FUNCTION_BLOCK FB_ParamMediatorWeu IMPLEMENTS I_ParamMediator
VAR
  _pCreateWorker : POINTER TO FB_WorkerDefGrid_Python;
  _pCamWorker : POINTER TO FB_WorkerDefGrid_Camera;
  _pDefWorker : POINTER TO FB_WorkerDefGrid_Deformation;
  bInitOk     : BOOL;
END_VAR

(*
  Release deformation ct
  TODO: find another way to do inter worker communication for generic methods.
*)
METHOD ClearCachedCT
VAR_INPUT
  iCT              : I_CT;
END_VAR
IF bInitOk THEN
  _pCreateWorker^.DeleteDefCt(iCT:=iCT);
END_IF
END_METHOD

(*
  Distance (Offset) from Master-Trigger to Master Reference Position.
  NOTE: This is normally the distance between the first (MASTER) StartPosDetection to first print Module (Printing Unit) 
*)
PROPERTY fMasterDetectToRefPos : LREAL
GET
IF bInitOk THEN
  fMasterDetectToRefPos := _pCamWorker^.fDetectToCamOffset + _pCamWorker^.fCameraToPrintOffset;
END_IF
END_GET
END_PROPERTY

METHOD init
VAR_INPUT
  pCreateWorker : POINTER TO FB_WorkerDefGrid_Python;
  pCamWorker : POINTER TO FB_WorkerDefGrid_Camera;
  pDefWorker : POINTER TO FB_WorkerDefGrid_Deformation;
END_VAR
IF pCamWorker <> 0 AND pCamWorker <>0 AND pCreateWorker <> 0 THEN
  _pCreateWorker := pCreateWorker;
  _pCamWorker := pCamWorker;
  _pDefWorker := pDefWorker;
  bInitOk := TRUE;
END_IF
END_METHOD

PROPERTY sCameraGridSettings : ST_CameraGridSettings
GET
IF bInitOk THEN
  sCameraGridSettings := _pCamWorker^.sCameraGridSettings;
END_IF
END_GET
END_PROPERTY

PROPERTY sDeformationGridSetttings : ST_DefGridSettings
GET
IF bInitOk THEN
  sDeformationGridSetttings := _pDefWorker^.sDeformationGridSettings;
END_IF
END_GET
END_PROPERTY

END_FUNCTION_BLOCK

(* stored: Version 1.1.0.1, ProductVersion 3.1.4024.11
   POU FB_ParamMediatorWeu: Id {30764c0e-d024-4e78-887c-61d747a091f1}, SpecialFunc None
   Folder I_ParamMediator: Id {a3f500e8-3f15-40d7-9c92-e10fd9ea2ea1}
   Method ClearCachedCT: Id {8e77280f-bf0a-46a8-8211-025431b5c21f}
   Property fMasterDetectToRefPos: Id {7f78ebba-c738-4eee-bd1f-29e6b7769eb8}
   Get Get: Id {19b38304-54a7-49bf-9679-1208bd51c285}
   Method init: Id {efdfd02d-5e3b-482c-bc07-2f8ffac60635}
   Property sCameraGridSettings: Id {fa75856d-5d24-4327-89a8-4ea8e08d9bd0}
   Get Get: Id {b9d9c9f7-6a09-4ee0-b36c-f72029ae80b6}
   Property sDeformationGridSetttings: Id {c3c33c61-5d1b-4422-8b45-ede2d3214c02}
   Get Get: Id {c9000730-0af4-4d84-9718-dd8d2b9b528d} *)
